FUNCTION Convert_REAL_TO_DT : BOOL
VAR_INPUT
	in : REAL;
	out : REFERENCE TO DT;
END_VAR
VAR
	converted : DT;
END_VAR

converted := REAL_TO_DT(in);

IF (DT_TO_REAL(converted) <> in) THEN
	RETURN;
END_IF

out := converted;
Convert_REAL_TO_DT := TRUE;

END_FUNCTION

(* stored: Version 1.1.0.1, ProductVersion 3.1.4024.12
   POU Convert_REAL_TO_DT: Id {87fd60d5-7223-4c82-ad83-5ba67edbb06a}, SpecialFunc None *)
